Staubli VAL3: getObjectLatch.pgx

public program getObjectLatch(num x_nConvNum (dimensions=1), num& x_nLatchedValue[] (dimensions=1), num& x_nError[] (dimensions=1))
  local point l_pPoint
begin
  // This program returns the encoder latched value of the object
  // that have been pushed into the buffer by the detection lib
  // of the specified conveyor.
  //
  // Input Param
  //  x_nConvNum  : Conveyor number
  //
  // Output Param
  //  x_nLatchedValue  : encoder latched value of the object
  //  x_nError         : Error code
  //    0 : No error
  //    1 : No data available
  //
  //----------------------------------------------------------------
  //
  switch x_nConvNum
    case 0
      call cnv0:getObjectLatch(x_nLatchedValue,x_nError)
    break
    case 1
      call cnv1:getObjectLatch(x_nLatchedValue,x_nError)
    break
  endSwitch
  //  if x_nError!=0
  //
  //  endIf
end
